{attribute 'qualified_only'}
{attribute 'strict'}
TYPE E_Event :
(
	Alarm := 0,
	Message := 1
);
END_TYPE

(* stored: Version 1.1.0.1, ProductVersion 3.1.4024.16
   DUT E_Event: Id {22d1da4b-378a-4de7-91ac-263413165b10} *)
